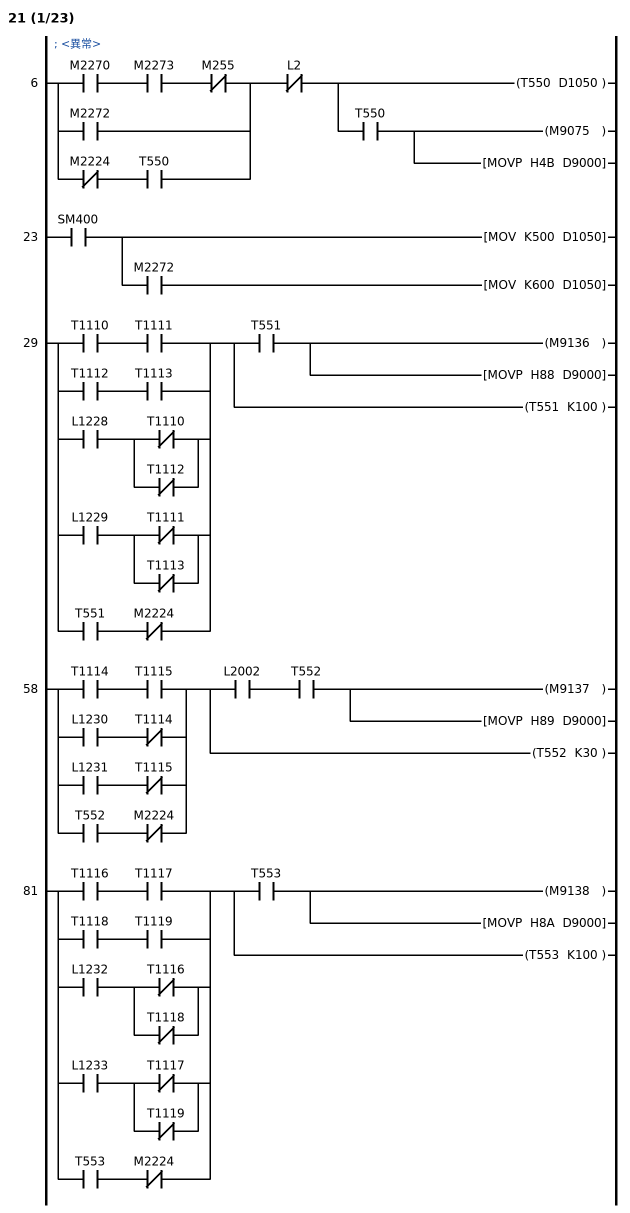
; <異常>
6     LD      M2270
      AND     M2273
      ANI     M255
      OR      M2272
      LDI     M2224
      AND     T550
      ORB
      ANI     L2
      OUT     T550 D1050
      AND     T550
      OUT     M9075
      MOVP    H4B D9000
23    LD      SM400
      MOV     K500 D1050
      AND     M2272
      MOV     K600 D1050
29    LD      T1110
      AND     T1111
      LD      T1112
      AND     T1113
      ORB
      LD      L1228
      LDI     T1110
      ORI     T1112
      ANB
      ORB
      LD      L1229
      LDI     T1111
      ORI     T1113
      ANB
      ORB
      LD      T551
      ANI     M2224
      ORB
      MPS
      AND     T551
      OUT     M9136
      MOVP    H88 D9000
      MPP
      OUT     T551 K100
58    LD      T1114
      AND     T1115
      LD      L1230
      ANI     T1114
      ORB
      LD      L1231
      ANI     T1115
      ORB
      LD      T552
      ANI     M2224
      ORB
      MPS
      AND     L2002
      AND     T552
      OUT     M9137
      MOVP    H89 D9000
      MPP
      OUT     T552 K30
81    LD      T1116
      AND     T1117
      LD      T1118
      AND     T1119
      ORB
      LD      L1232
      LDI     T1116
      ORI     T1118
      ANB
      ORB
      LD      L1233
      LDI     T1117
      ORI     T1119
      ANB
      ORB
      LD      T553
      ANI     M2224
      ORB
      MPS
      AND     T553
      OUT     M9138
      MOVP    H8A D9000
      MPP
      OUT     T553 K100
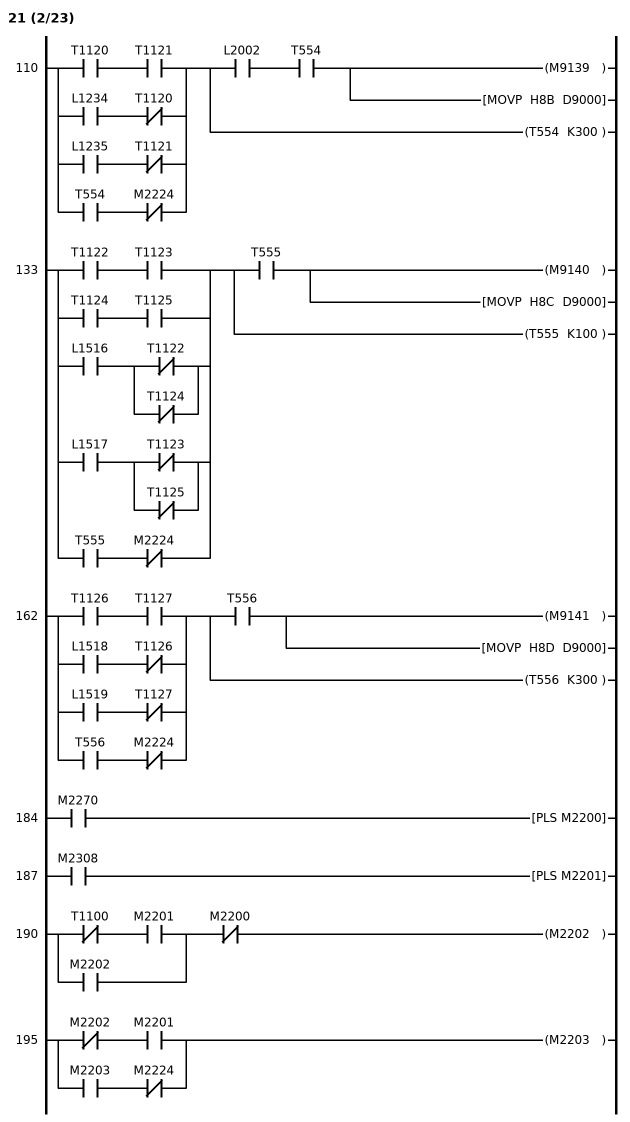
110   LD      T1120
      AND     T1121
      LD      L1234
      ANI     T1120
      ORB
      LD      L1235
      ANI     T1121
      ORB
      LD      T554
      ANI     M2224
      ORB
      MPS
      AND     L2002
      AND     T554
      OUT     M9139
      MOVP    H8B D9000
      MPP
      OUT     T554 K300
133   LD      T1122
      AND     T1123
      LD      T1124
      AND     T1125
      ORB
      LD      L1516
      LDI     T1122
      ORI     T1124
      ANB
      ORB
      LD      L1517
      LDI     T1123
      ORI     T1125
      ANB
      ORB
      LD      T555
      ANI     M2224
      ORB
      MPS
      AND     T555
      OUT     M9140
      MOVP    H8C D9000
      MPP
      OUT     T555 K100
162   LD      T1126
      AND     T1127
      LD      L1518
      ANI     T1126
      ORB
      LD      L1519
      ANI     T1127
      ORB
      LD      T556
      ANI     M2224
      ORB
      MPS
      AND     T556
      OUT     M9141
      MOVP    H8D D9000
      MPP
      OUT     T556 K300
184   LD      M2270
      PLS     M2200
187   LD      M2308
      PLS     M2201
190   LDI     T1100
      AND     M2201
      OR      M2202
      ANI     M2200
      OUT     M2202
195   LDI     M2202
      AND     M2201
      LD      M2203
      ANI     M2224
      ORB
      OUT     M2203
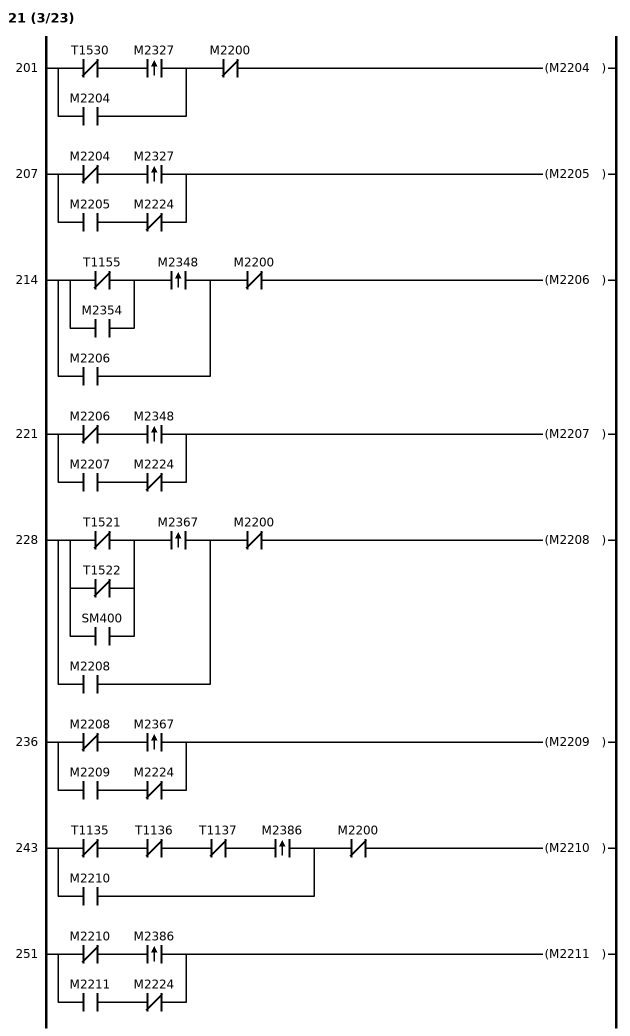
201   LDI     T1530
      ANDP    M2327
      OR      M2204
      ANI     M2200
      OUT     M2204
207   LDI     M2204
      ANDP    M2327
      LD      M2205
      ANI     M2224
      ORB
      OUT     M2205
214   LDI     T1155
      OR      M2354
      ANDP    M2348
      OR      M2206
      ANI     M2200
      OUT     M2206
221   LDI     M2206
      ANDP    M2348
      LD      M2207
      ANI     M2224
      ORB
      OUT     M2207
228   LDI     T1521
      ORI     T1522
      OR      SM400
      ANDP    M2367
      OR      M2208
      ANI     M2200
      OUT     M2208
236   LDI     M2208
      ANDP    M2367
      LD      M2209
      ANI     M2224
      ORB
      OUT     M2209
243   LDI     T1135
      ANI     T1136
      ANI     T1137
      ANDP    M2386
      OR      M2210
      ANI     M2200
      OUT     M2210
251   LDI     M2210
      ANDP    M2386
      LD      M2211
      ANI     M2224
      ORB
      OUT     M2211
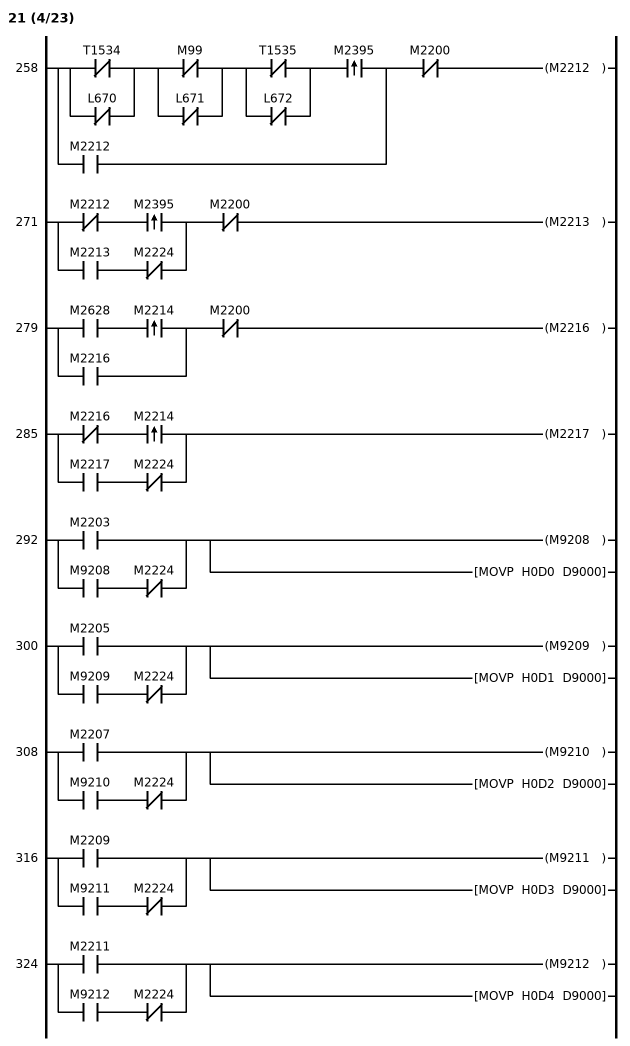
258   LDI     T1534
      ORI     L670
      LDI     M99
      ORI     L671
      ANB
      LDI     T1535
      ORI     L672
      ANB
      ANDP    M2395
      OR      M2212
      ANI     M2200
      OUT     M2212
271   LDI     M2212
      ANDP    M2395
      LD      M2213
      ANI     M2224
      ORB
      ANI     M2200
      OUT     M2213
279   LD      M2628
      ANDP    M2214
      OR      M2216
      ANI     M2200
      OUT     M2216
285   LDI     M2216
      ANDP    M2214
      LD      M2217
      ANI     M2224
      ORB
      OUT     M2217
292   LD      M2203
      LD      M9208
      ANI     M2224
      ORB
      OUT     M9208
      MOVP    H0D0 D9000
300   LD      M2205
      LD      M9209
      ANI     M2224
      ORB
      OUT     M9209
      MOVP    H0D1 D9000
308   LD      M2207
      LD      M9210
      ANI     M2224
      ORB
      OUT     M9210
      MOVP    H0D2 D9000
316   LD      M2209
      LD      M9211
      ANI     M2224
      ORB
      OUT     M9211
      MOVP    H0D3 D9000
324   LD      M2211
      LD      M9212
      ANI     M2224
      ORB
      OUT     M9212
      MOVP    H0D4 D9000
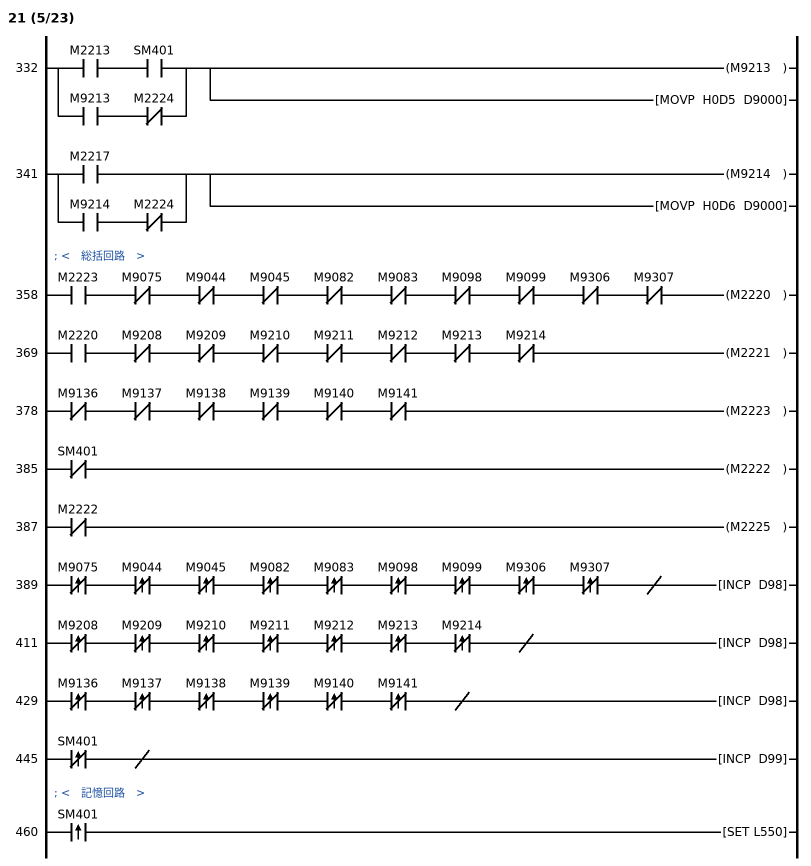
332   LD      M2213
      AND     SM401
      LD      M9213
      ANI     M2224
      ORB
      OUT     M9213
      MOVP    H0D5 D9000
341   LD      M2217
      LD      M9214
      ANI     M2224
      ORB
      OUT     M9214
      MOVP    H0D6 D9000
; <　総括回路　>
358   LD      M2223
      ANI     M9075
      ANI     M9044
      ANI     M9045
      ANI     M9082
      ANI     M9083
      ANI     M9098
      ANI     M9099
      ANI     M9306
      ANI     M9307
      OUT     M2220
369   LD      M2220
      ANI     M9208
      ANI     M9209
      ANI     M9210
      ANI     M9211
      ANI     M9212
      ANI     M9213
      ANI     M9214
      OUT     M2221
378   LDI     M9136
      ANI     M9137
      ANI     M9138
      ANI     M9139
      ANI     M9140
      ANI     M9141
      OUT     M2223
385   LDI     SM401
      OUT     M2222
387   LDI     M2222
      OUT     M2225
389   LDPI    M9075
      ANDPI   M9044
      ANDPI   M9045
      ANDPI   M9082
      ANDPI   M9083
      ANDPI   M9098
      ANDPI   M9099
      ANDPI   M9306
      ANDPI   M9307
      INV
      INCP    D98
411   LDPI    M9208
      ANDPI   M9209
      ANDPI   M9210
      ANDPI   M9211
      ANDPI   M9212
      ANDPI   M9213
      ANDPI   M9214
      INV
      INCP    D98
429   LDPI    M9136
      ANDPI   M9137
      ANDPI   M9138
      ANDPI   M9139
      ANDPI   M9140
      ANDPI   M9141
      INV
      INCP    D98
445   LDPI    SM401
      INV
      INCP    D99
; <　記憶回路　>
460   LDP     SM401
      SET     L550
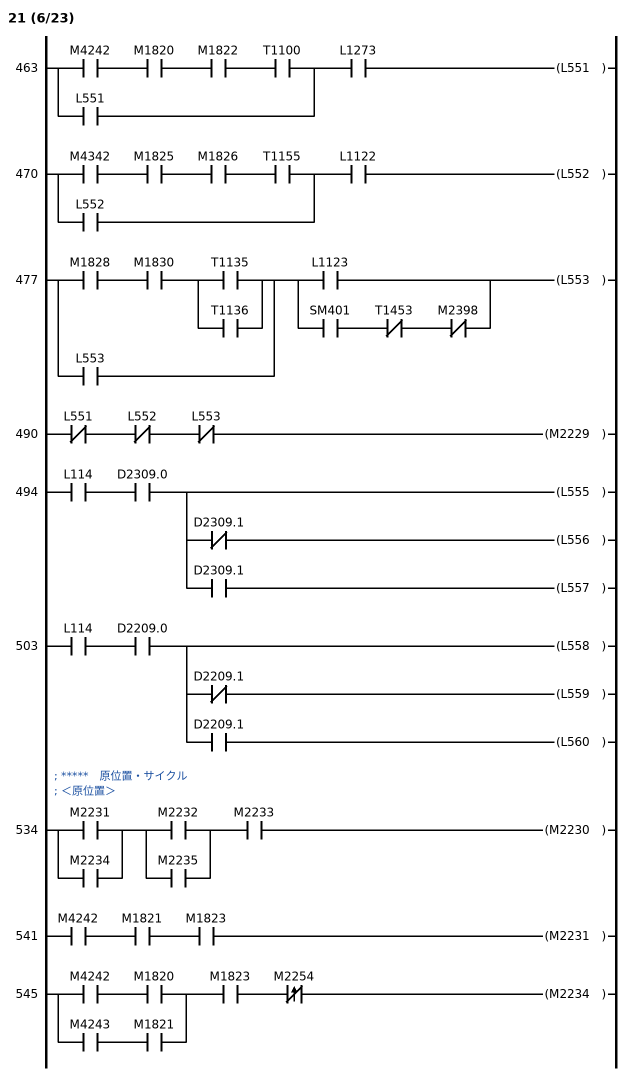
463   LD      M4242
      AND     M1820
      AND     M1822
      AND     T1100
      OR      L551
      AND     L1273
      OUT     L551
470   LD      M4342
      AND     M1825
      AND     M1826
      AND     T1155
      OR      L552
      AND     L1122
      OUT     L552
477   LD      M1828
      AND     M1830
      LD      T1135
      OR      T1136
      ANB
      OR      L553
      LD      L1123
      LD      SM401
      ANI     T1453
      ANI     M2398
      ORB
      ANB
      OUT     L553
490   LDI     L551
      ANI     L552
      ANI     L553
      OUT     M2229
494   LD      L114
      AND     D2309.0
      OUT     L555
      MPS
      ANI     D2309.1
      OUT     L556
      MPP
      AND     D2309.1
      OUT     L557
503   LD      L114
      AND     D2209.0
      OUT     L558
      MPS
      ANI     D2209.1
      OUT     L559
      MPP
      AND     D2209.1
      OUT     L560
; *****　原位置・サイクル
; ＜原位置＞
534   LD      M2231
      OR      M2234
      LD      M2232
      OR      M2235
      ANB
      AND     M2233
      OUT     M2230
541   LD      M4242
      AND     M1821
      AND     M1823
      OUT     M2231
545   LD      M4242
      AND     M1820
      LD      M4243
      AND     M1821
      ORB
      AND     M1823
      ANDPI   M2254
      OUT     M2234
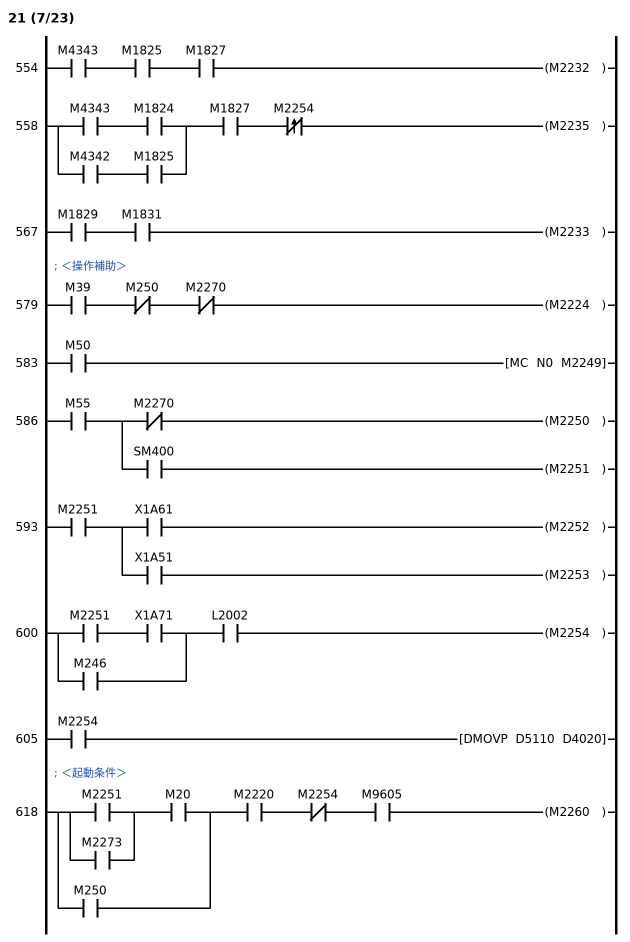
554   LD      M4343
      AND     M1825
      AND     M1827
      OUT     M2232
558   LD      M4343
      AND     M1824
      LD      M4342
      AND     M1825
      ORB
      AND     M1827
      ANDPI   M2254
      OUT     M2235
567   LD      M1829
      AND     M1831
      OUT     M2233
; ＜操作補助＞
579   LD      M39
      ANI     M250
      ANI     M2270
      OUT     M2224
583   LD      M50
      MC      N0 M2249
586   LD      M55
      MPS
      ANI     M2270
      OUT     M2250
      MPP
      AND     SM400
      OUT     M2251
593   LD      M2251
      MPS
      AND     X1A61
      OUT     M2252
      MPP
      AND     X1A51
      OUT     M2253
600   LD      M2251
      AND     X1A71
      OR      M246
      AND     L2002
      OUT     M2254
605   LD      M2254
      DMOVP   D5110 D4020
; ＜起動条件＞
618   LD      M2251
      OR      M2273
      AND     M20
      OR      M250
      AND     M2220
      ANI     M2254
      AND     M9605
      OUT     M2260
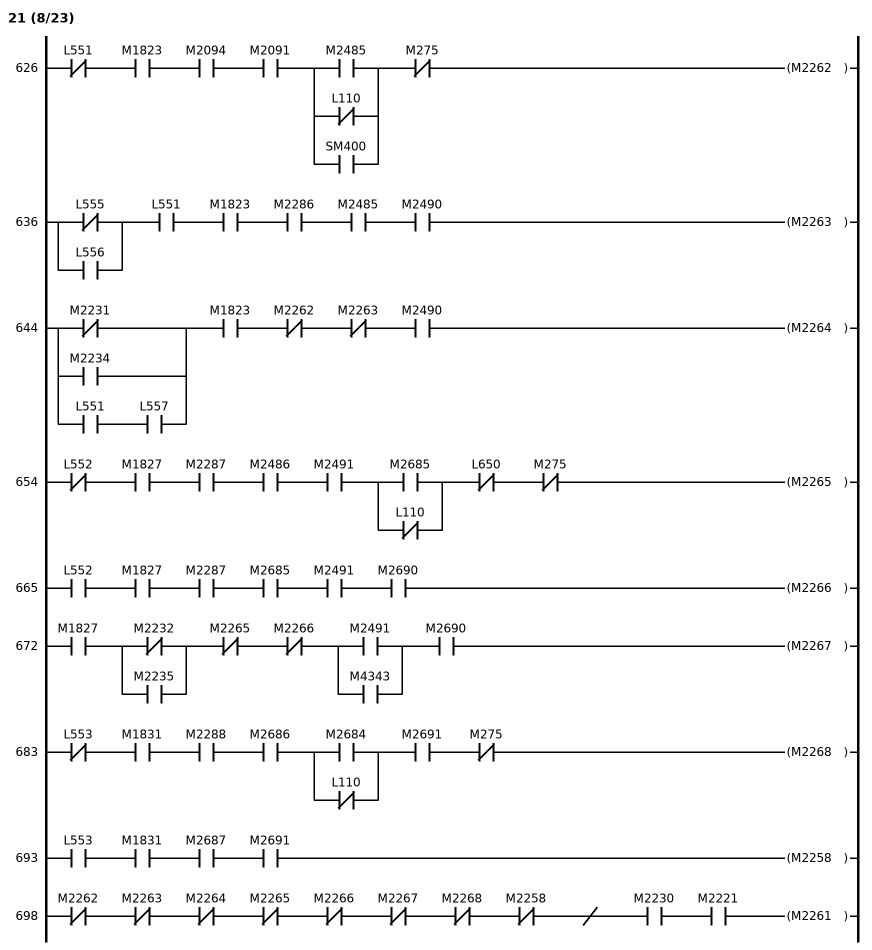
626   LDI     L551
      AND     M1823
      AND     M2094
      AND     M2091
      LD      M2485
      ORI     L110
      OR      SM400
      ANB
      ANI     M275
      OUT     M2262
636   LDI     L555
      OR      L556
      AND     L551
      AND     M1823
      AND     M2286
      AND     M2485
      AND     M2490
      OUT     M2263
644   LDI     M2231
      OR      M2234
      LD      L551
      AND     L557
      ORB
      AND     M1823
      ANI     M2262
      ANI     M2263
      AND     M2490
      OUT     M2264
654   LDI     L552
      AND     M1827
      AND     M2287
      AND     M2486
      AND     M2491
      LD      M2685
      ORI     L110
      ANB
      ANI     L650
      ANI     M275
      OUT     M2265
665   LD      L552
      AND     M1827
      AND     M2287
      AND     M2685
      AND     M2491
      AND     M2690
      OUT     M2266
672   LD      M1827
      LDI     M2232
      OR      M2235
      ANB
      ANI     M2265
      ANI     M2266
      LD      M2491
      OR      M4343
      ANB
      AND     M2690
      OUT     M2267
683   LDI     L553
      AND     M1831
      AND     M2288
      AND     M2686
      LD      M2684
      ORI     L110
      ANB
      AND     M2691
      ANI     M275
      OUT     M2268
693   LD      L553
      AND     M1831
      AND     M2687
      AND     M2691
      OUT     M2258
698   LDI     M2262
      ANI     M2263
      ANI     M2264
      ANI     M2265
      ANI     M2266
      ANI     M2267
      ANI     M2268
      ANI     M2258
      INV
      AND     M2230
      AND     M2221
      OUT     M2261
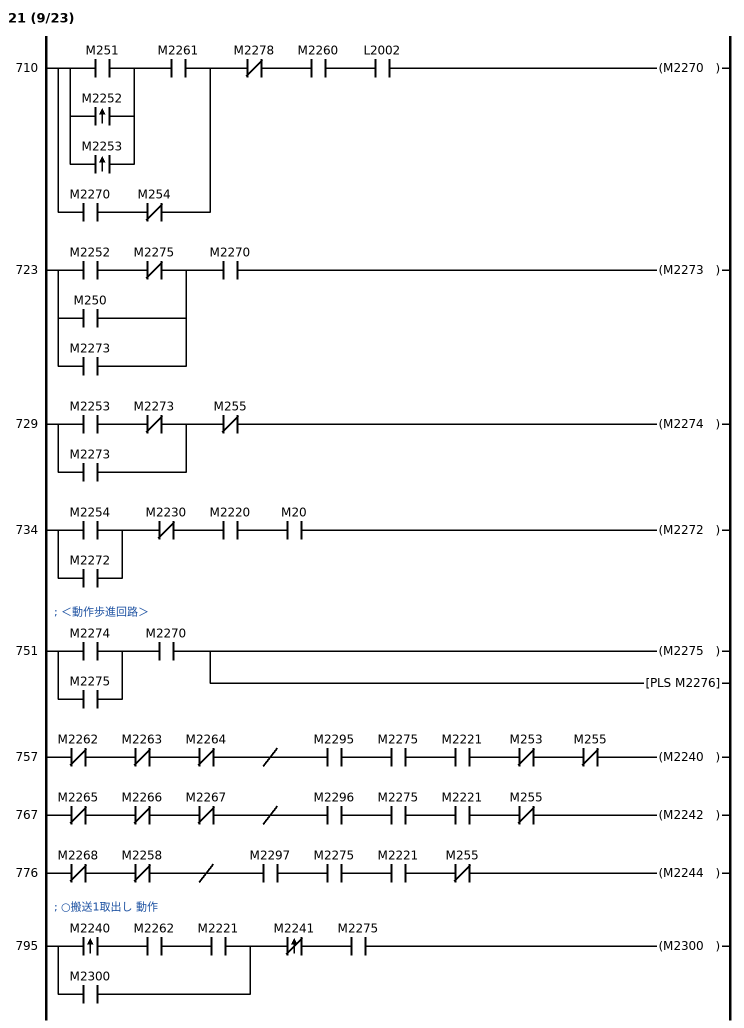
710   LD      M251
      ORP     M2252
      ORP     M2253
      AND     M2261
      LD      M2270
      ANI     M254
      ORB
      ANI     M2278
      AND     M2260
      AND     L2002
      OUT     M2270
723   LD      M2252
      ANI     M2275
      OR      M250
      OR      M2273
      AND     M2270
      OUT     M2273
729   LD      M2253
      ANI     M2273
      OR      M2273
      ANI     M255
      OUT     M2274
734   LD      M2254
      OR      M2272
      ANI     M2230
      AND     M2220
      AND     M20
      OUT     M2272
; ＜動作歩進回路＞
751   LD      M2274
      OR      M2275
      AND     M2270
      OUT     M2275
      PLS     M2276
757   LDI     M2262
      ANI     M2263
      ANI     M2264
      INV
      AND     M2295
      AND     M2275
      AND     M2221
      ANI     M253
      ANI     M255
      OUT     M2240
767   LDI     M2265
      ANI     M2266
      ANI     M2267
      INV
      AND     M2296
      AND     M2275
      AND     M2221
      ANI     M255
      OUT     M2242
776   LDI     M2268
      ANI     M2258
      INV
      AND     M2297
      AND     M2275
      AND     M2221
      ANI     M255
      OUT     M2244
; ○搬送1取出し 動作
795   LDP     M2240
      AND     M2262
      AND     M2221
      OR      M2300
      ANDPI   M2241
      AND     M2275
      OUT     M2300
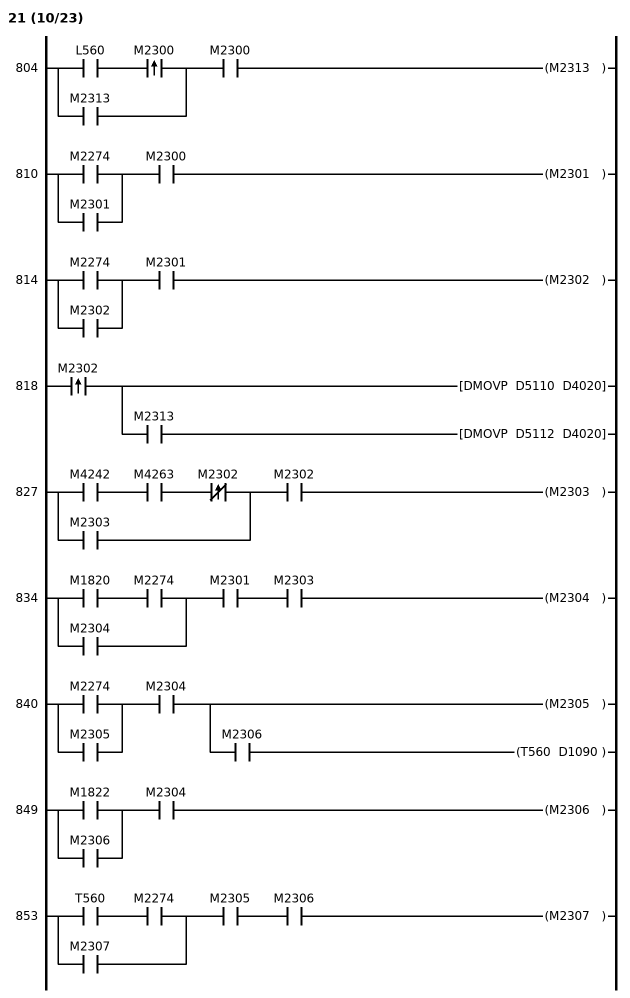
804   LD      L560
      ANDP    M2300
      OR      M2313
      AND     M2300
      OUT     M2313
810   LD      M2274
      OR      M2301
      AND     M2300
      OUT     M2301
814   LD      M2274
      OR      M2302
      AND     M2301
      OUT     M2302
818   LDP     M2302
      DMOVP   D5110 D4020
      AND     M2313
      DMOVP   D5112 D4020
827   LD      M4242
      AND     M4263
      ANDPI   M2302
      OR      M2303
      AND     M2302
      OUT     M2303
834   LD      M1820
      AND     M2274
      OR      M2304
      AND     M2301
      AND     M2303
      OUT     M2304
840   LD      M2274
      OR      M2305
      AND     M2304
      OUT     M2305
      AND     M2306
      OUT     T560 D1090
849   LD      M1822
      OR      M2306
      AND     M2304
      OUT     M2306
853   LD      T560
      AND     M2274
      OR      M2307
      AND     M2305
      AND     M2306
      OUT     M2307
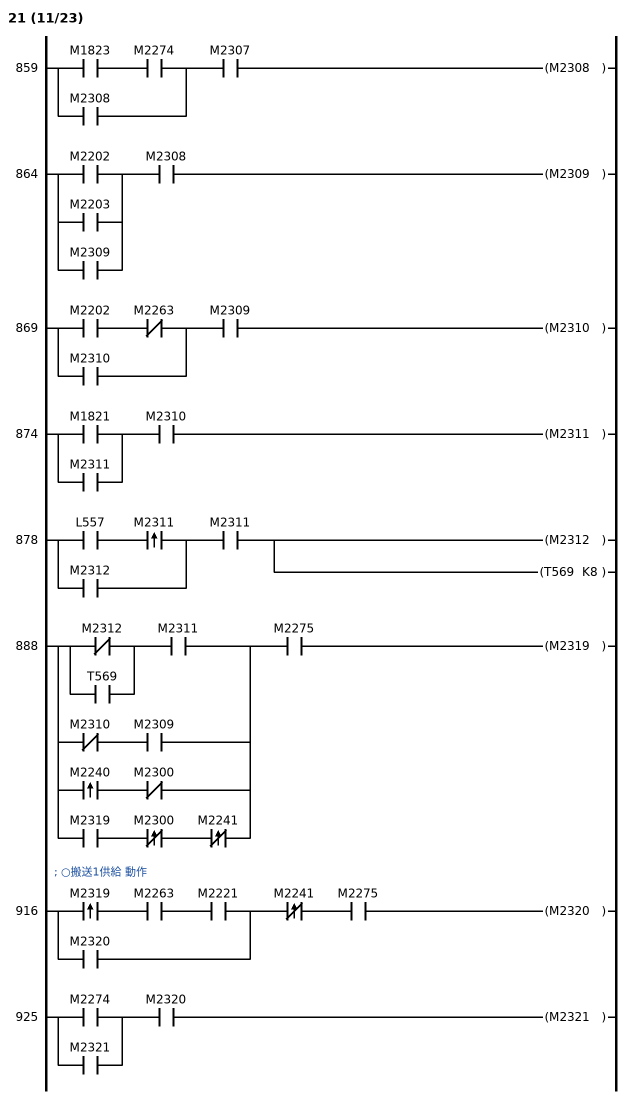
859   LD      M1823
      AND     M2274
      OR      M2308
      AND     M2307
      OUT     M2308
864   LD      M2202
      OR      M2203
      OR      M2309
      AND     M2308
      OUT     M2309
869   LD      M2202
      ANI     M2263
      OR      M2310
      AND     M2309
      OUT     M2310
874   LD      M1821
      OR      M2311
      AND     M2310
      OUT     M2311
878   LD      L557
      ANDP    M2311
      OR      M2312
      AND     M2311
      OUT     M2312
      OUT     T569 K8
888   LDI     M2312
      OR      T569
      AND     M2311
      LDI     M2310
      AND     M2309
      ORB
      LDP     M2240
      ANI     M2300
      ORB
      LD      M2319
      ANDPI   M2300
      ANDPI   M2241
      ORB
      AND     M2275
      OUT     M2319
; ○搬送1供給 動作
916   LDP     M2319
      AND     M2263
      AND     M2221
      OR      M2320
      ANDPI   M2241
      AND     M2275
      OUT     M2320
925   LD      M2274
      OR      M2321
      AND     M2320
      OUT     M2321
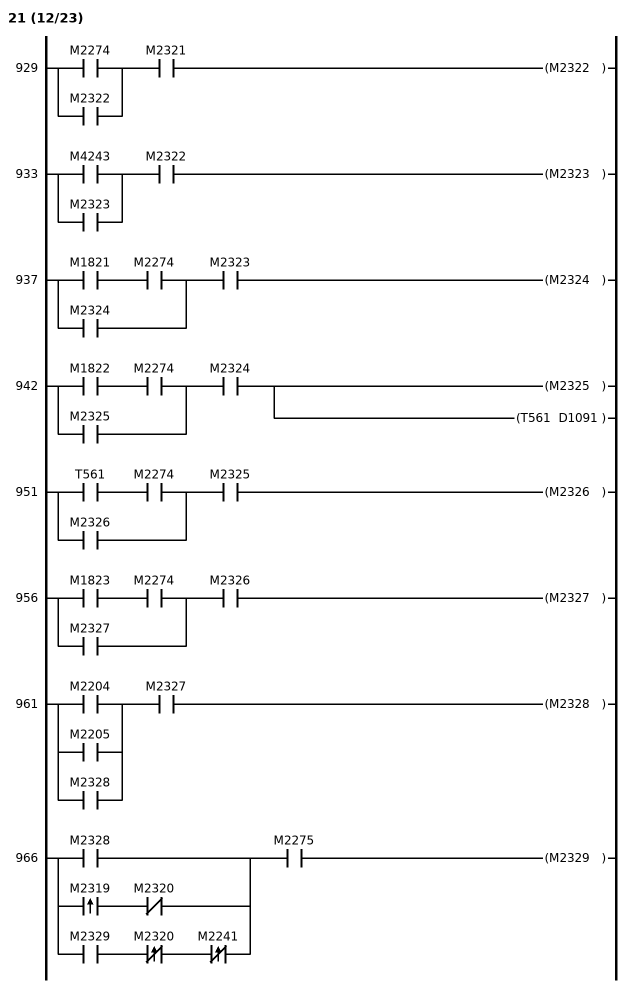
929   LD      M2274
      OR      M2322
      AND     M2321
      OUT     M2322
933   LD      M4243
      OR      M2323
      AND     M2322
      OUT     M2323
937   LD      M1821
      AND     M2274
      OR      M2324
      AND     M2323
      OUT     M2324
942   LD      M1822
      AND     M2274
      OR      M2325
      AND     M2324
      OUT     M2325
      OUT     T561 D1091
951   LD      T561
      AND     M2274
      OR      M2326
      AND     M2325
      OUT     M2326
956   LD      M1823
      AND     M2274
      OR      M2327
      AND     M2326
      OUT     M2327
961   LD      M2204
      OR      M2205
      OR      M2328
      AND     M2327
      OUT     M2328
966   LD      M2328
      LDP     M2319
      ANI     M2320
      ORB
      LD      M2329
      ANDPI   M2320
      ANDPI   M2241
      ORB
      AND     M2275
      OUT     M2329
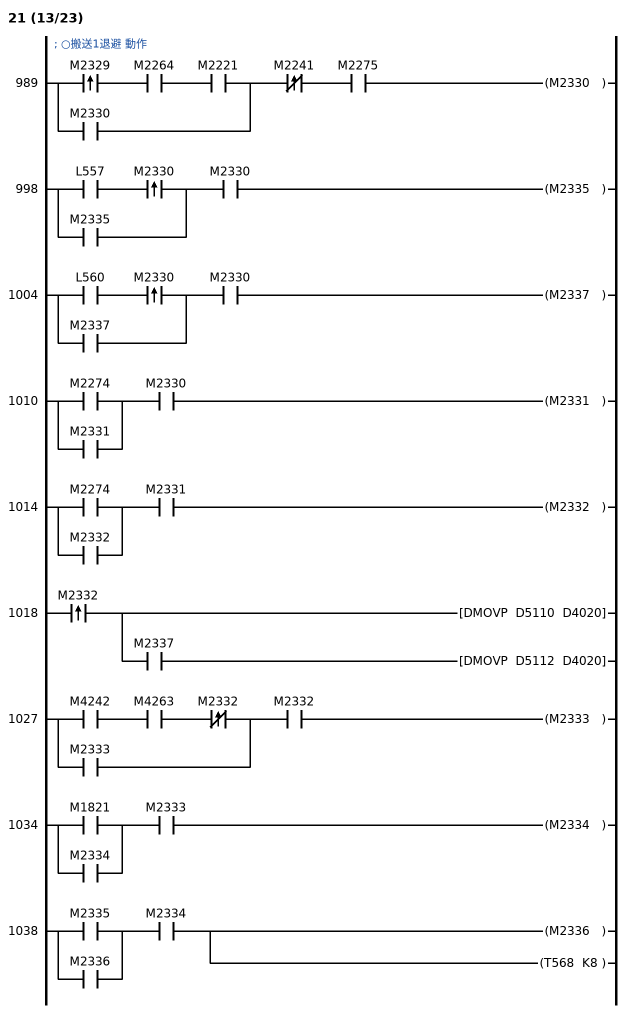
; ○搬送1退避 動作
989   LDP     M2329
      AND     M2264
      AND     M2221
      OR      M2330
      ANDPI   M2241
      AND     M2275
      OUT     M2330
998   LD      L557
      ANDP    M2330
      OR      M2335
      AND     M2330
      OUT     M2335
1004  LD      L560
      ANDP    M2330
      OR      M2337
      AND     M2330
      OUT     M2337
1010  LD      M2274
      OR      M2331
      AND     M2330
      OUT     M2331
1014  LD      M2274
      OR      M2332
      AND     M2331
      OUT     M2332
1018  LDP     M2332
      DMOVP   D5110 D4020
      AND     M2337
      DMOVP   D5112 D4020
1027  LD      M4242
      AND     M4263
      ANDPI   M2332
      OR      M2333
      AND     M2332
      OUT     M2333
1034  LD      M1821
      OR      M2334
      AND     M2333
      OUT     M2334
1038  LD      M2335
      OR      M2336
      AND     M2334
      OUT     M2336
      OUT     T568 K8
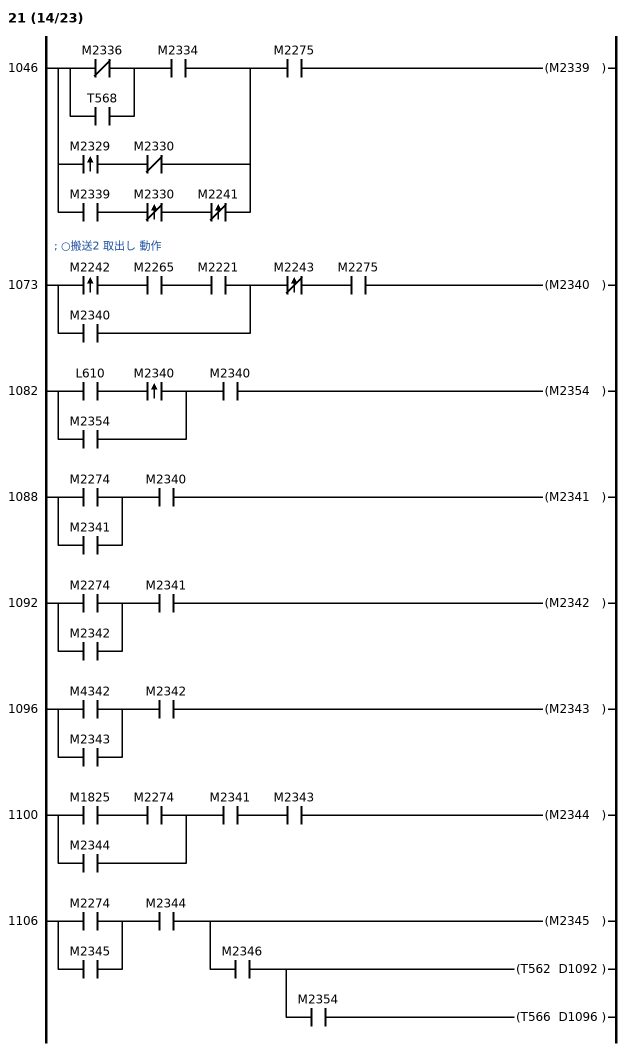
1046  LDI     M2336
      OR      T568
      AND     M2334
      LDP     M2329
      ANI     M2330
      ORB
      LD      M2339
      ANDPI   M2330
      ANDPI   M2241
      ORB
      AND     M2275
      OUT     M2339
; ○搬送2 取出し 動作
1073  LDP     M2242
      AND     M2265
      AND     M2221
      OR      M2340
      ANDPI   M2243
      AND     M2275
      OUT     M2340
1082  LD      L610
      ANDP    M2340
      OR      M2354
      AND     M2340
      OUT     M2354
1088  LD      M2274
      OR      M2341
      AND     M2340
      OUT     M2341
1092  LD      M2274
      OR      M2342
      AND     M2341
      OUT     M2342
1096  LD      M4342
      OR      M2343
      AND     M2342
      OUT     M2343
1100  LD      M1825
      AND     M2274
      OR      M2344
      AND     M2341
      AND     M2343
      OUT     M2344
1106  LD      M2274
      OR      M2345
      AND     M2344
      OUT     M2345
      AND     M2346
      OUT     T562 D1092
      AND     M2354
      OUT     T566 D1096
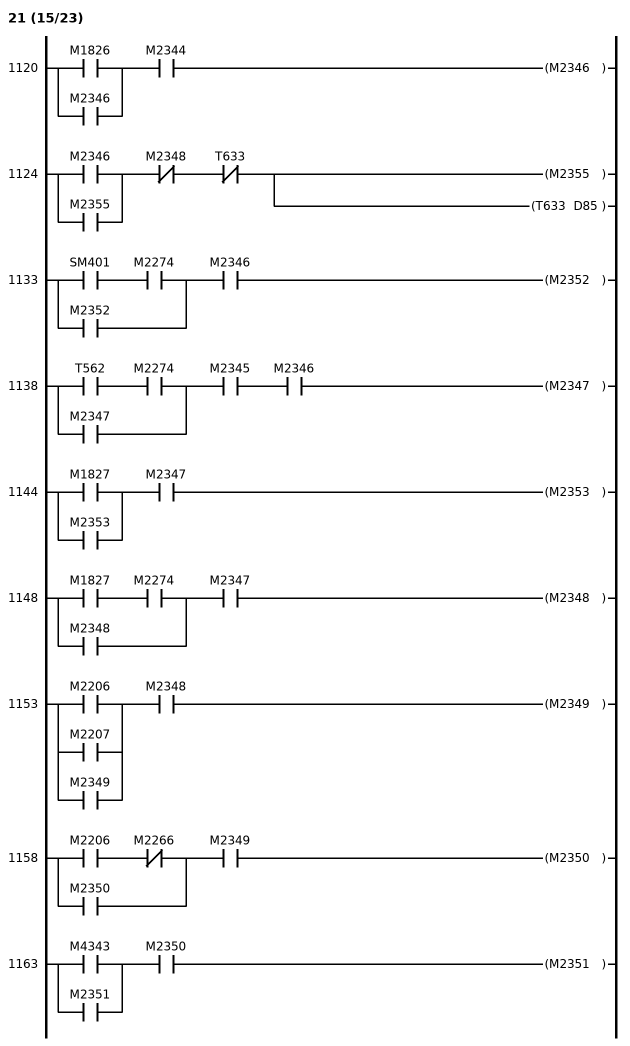
1120  LD      M1826
      OR      M2346
      AND     M2344
      OUT     M2346
1124  LD      M2346
      OR      M2355
      ANI     M2348
      ANI     T633
      OUT     M2355
      OUT     T633 D85
1133  LD      SM401
      AND     M2274
      OR      M2352
      AND     M2346
      OUT     M2352
1138  LD      T562
      AND     M2274
      OR      M2347
      AND     M2345
      AND     M2346
      OUT     M2347
1144  LD      M1827
      OR      M2353
      AND     M2347
      OUT     M2353
1148  LD      M1827
      AND     M2274
      OR      M2348
      AND     M2347
      OUT     M2348
1153  LD      M2206
      OR      M2207
      OR      M2349
      AND     M2348
      OUT     M2349
1158  LD      M2206
      ANI     M2266
      OR      M2350
      AND     M2349
      OUT     M2350
1163  LD      M4343
      OR      M2351
      AND     M2350
      OUT     M2351
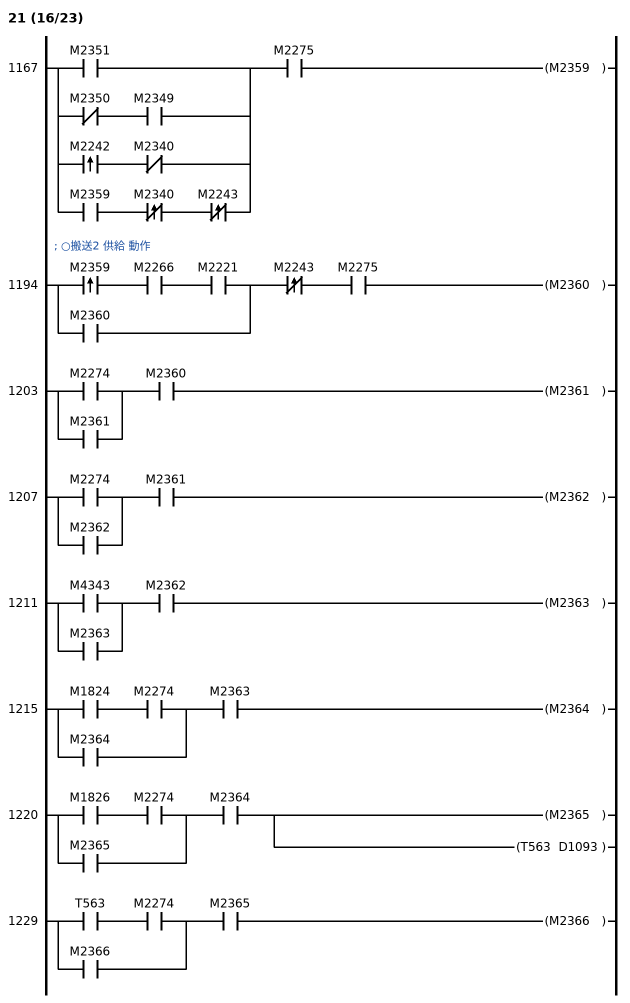
1167  LD      M2351
      LDI     M2350
      AND     M2349
      ORB
      LDP     M2242
      ANI     M2340
      ORB
      LD      M2359
      ANDPI   M2340
      ANDPI   M2243
      ORB
      AND     M2275
      OUT     M2359
; ○搬送2 供給 動作
1194  LDP     M2359
      AND     M2266
      AND     M2221
      OR      M2360
      ANDPI   M2243
      AND     M2275
      OUT     M2360
1203  LD      M2274
      OR      M2361
      AND     M2360
      OUT     M2361
1207  LD      M2274
      OR      M2362
      AND     M2361
      OUT     M2362
1211  LD      M4343
      OR      M2363
      AND     M2362
      OUT     M2363
1215  LD      M1824
      AND     M2274
      OR      M2364
      AND     M2363
      OUT     M2364
1220  LD      M1826
      AND     M2274
      OR      M2365
      AND     M2364
      OUT     M2365
      OUT     T563 D1093
1229  LD      T563
      AND     M2274
      OR      M2366
      AND     M2365
      OUT     M2366
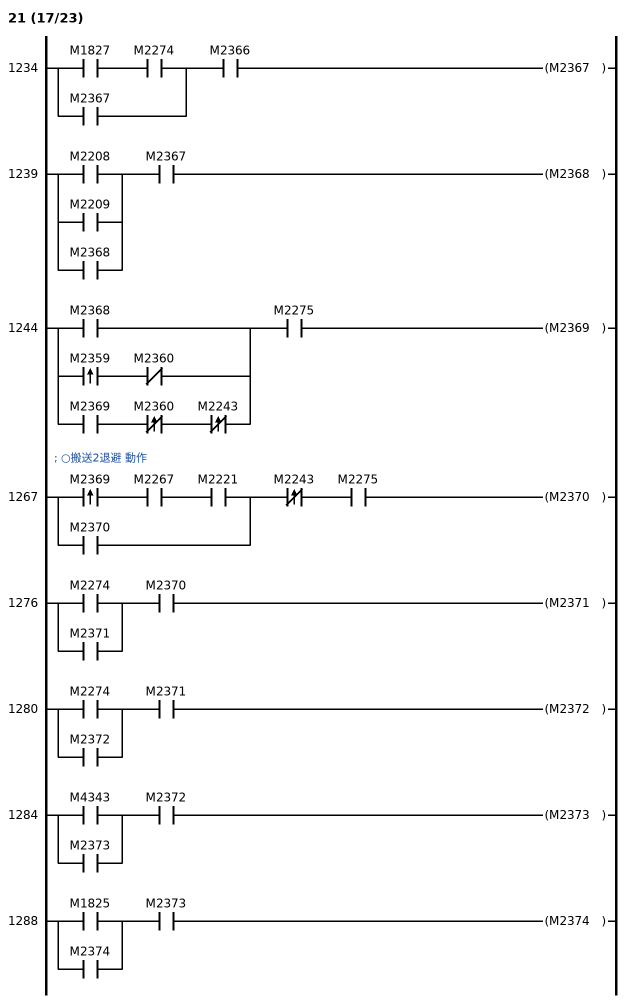
1234  LD      M1827
      AND     M2274
      OR      M2367
      AND     M2366
      OUT     M2367
1239  LD      M2208
      OR      M2209
      OR      M2368
      AND     M2367
      OUT     M2368
1244  LD      M2368
      LDP     M2359
      ANI     M2360
      ORB
      LD      M2369
      ANDPI   M2360
      ANDPI   M2243
      ORB
      AND     M2275
      OUT     M2369
; ○搬送2退避 動作
1267  LDP     M2369
      AND     M2267
      AND     M2221
      OR      M2370
      ANDPI   M2243
      AND     M2275
      OUT     M2370
1276  LD      M2274
      OR      M2371
      AND     M2370
      OUT     M2371
1280  LD      M2274
      OR      M2372
      AND     M2371
      OUT     M2372
1284  LD      M4343
      OR      M2373
      AND     M2372
      OUT     M2373
1288  LD      M1825
      OR      M2374
      AND     M2373
      OUT     M2374
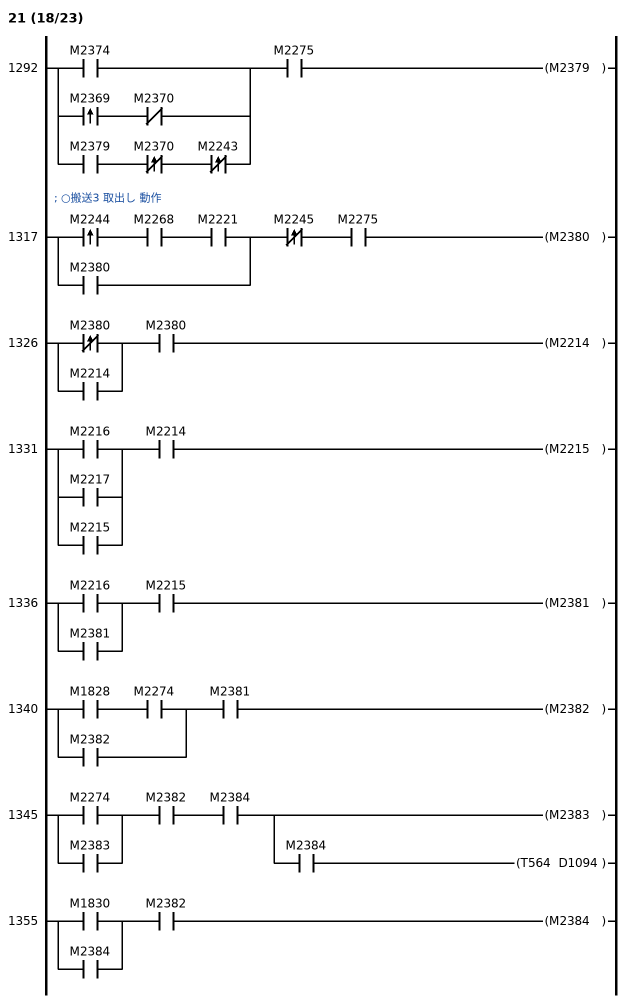
1292  LD      M2374
      LDP     M2369
      ANI     M2370
      ORB
      LD      M2379
      ANDPI   M2370
      ANDPI   M2243
      ORB
      AND     M2275
      OUT     M2379
; ○搬送3 取出し 動作
1317  LDP     M2244
      AND     M2268
      AND     M2221
      OR      M2380
      ANDPI   M2245
      AND     M2275
      OUT     M2380
1326  LDPI    M2380
      OR      M2214
      AND     M2380
      OUT     M2214
1331  LD      M2216
      OR      M2217
      OR      M2215
      AND     M2214
      OUT     M2215
1336  LD      M2216
      OR      M2381
      AND     M2215
      OUT     M2381
1340  LD      M1828
      AND     M2274
      OR      M2382
      AND     M2381
      OUT     M2382
1345  LD      M2274
      OR      M2383
      AND     M2382
      AND     M2384
      OUT     M2383
      AND     M2384
      OUT     T564 D1094
1355  LD      M1830
      OR      M2384
      AND     M2382
      OUT     M2384
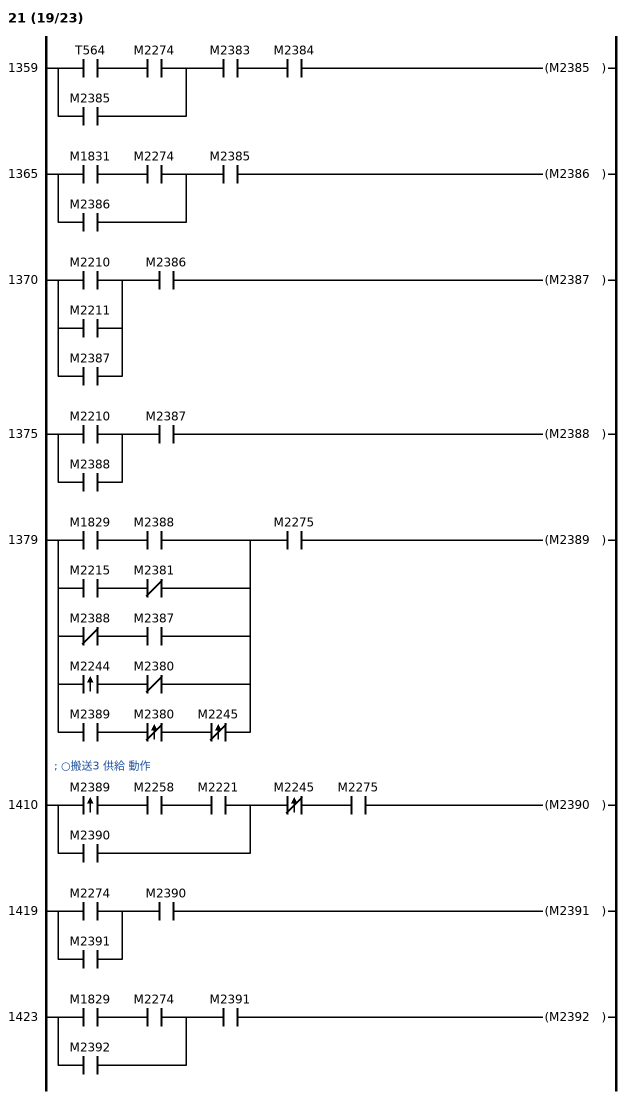
1359  LD      T564
      AND     M2274
      OR      M2385
      AND     M2383
      AND     M2384
      OUT     M2385
1365  LD      M1831
      AND     M2274
      OR      M2386
      AND     M2385
      OUT     M2386
1370  LD      M2210
      OR      M2211
      OR      M2387
      AND     M2386
      OUT     M2387
1375  LD      M2210
      OR      M2388
      AND     M2387
      OUT     M2388
1379  LD      M1829
      AND     M2388
      LD      M2215
      ANI     M2381
      ORB
      LDI     M2388
      AND     M2387
      ORB
      LDP     M2244
      ANI     M2380
      ORB
      LD      M2389
      ANDPI   M2380
      ANDPI   M2245
      ORB
      AND     M2275
      OUT     M2389
; ○搬送3 供給 動作
1410  LDP     M2389
      AND     M2258
      AND     M2221
      OR      M2390
      ANDPI   M2245
      AND     M2275
      OUT     M2390
1419  LD      M2274
      OR      M2391
      AND     M2390
      OUT     M2391
1423  LD      M1829
      AND     M2274
      OR      M2392
      AND     M2391
      OUT     M2392
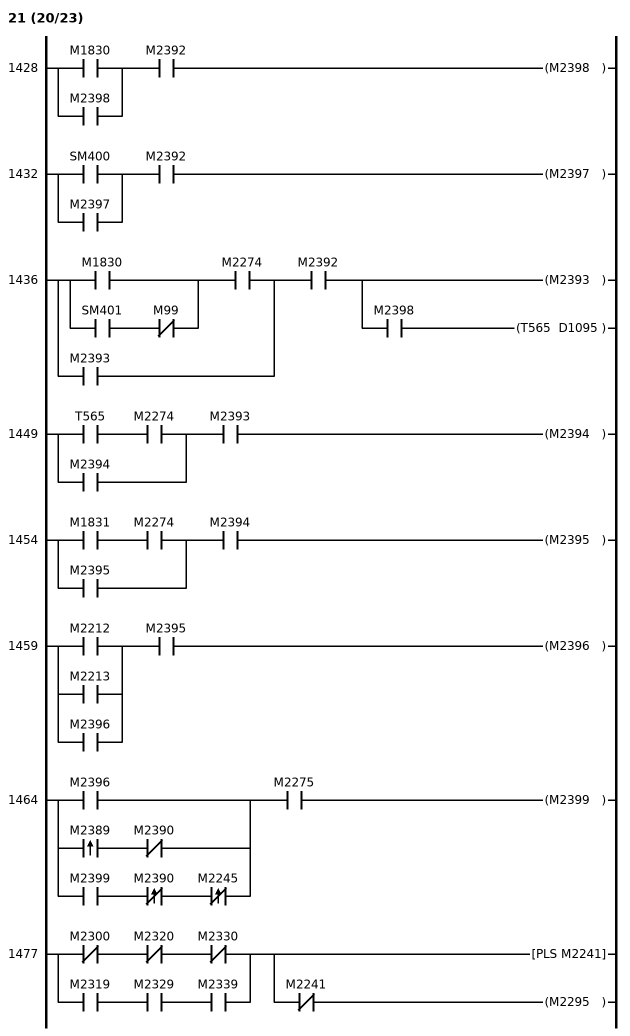
1428  LD      M1830
      OR      M2398
      AND     M2392
      OUT     M2398
1432  LD      SM400
      OR      M2397
      AND     M2392
      OUT     M2397
1436  LD      M1830
      LD      SM401
      ANI     M99
      ORB
      AND     M2274
      OR      M2393
      AND     M2392
      OUT     M2393
      AND     M2398
      OUT     T565 D1095
1449  LD      T565
      AND     M2274
      OR      M2394
      AND     M2393
      OUT     M2394
1454  LD      M1831
      AND     M2274
      OR      M2395
      AND     M2394
      OUT     M2395
1459  LD      M2212
      OR      M2213
      OR      M2396
      AND     M2395
      OUT     M2396
1464  LD      M2396
      LDP     M2389
      ANI     M2390
      ORB
      LD      M2399
      ANDPI   M2390
      ANDPI   M2245
      ORB
      AND     M2275
      OUT     M2399
1477  LDI     M2300
      ANI     M2320
      ANI     M2330
      LD      M2319
      AND     M2329
      AND     M2339
      ORB
      PLS     M2241
      ANI     M2241
      OUT     M2295
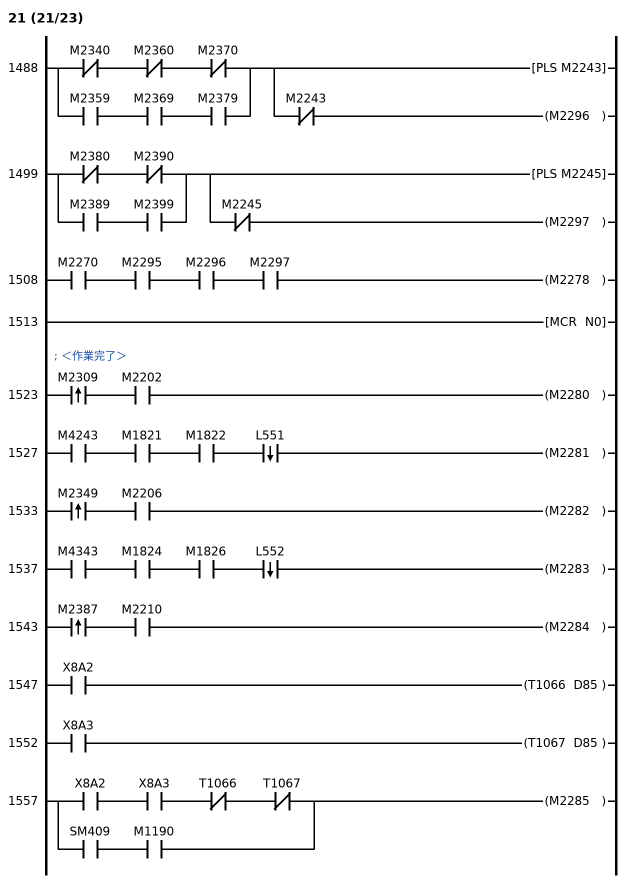
1488  LDI     M2340
      ANI     M2360
      ANI     M2370
      LD      M2359
      AND     M2369
      AND     M2379
      ORB
      PLS     M2243
      ANI     M2243
      OUT     M2296
1499  LDI     M2380
      ANI     M2390
      LD      M2389
      AND     M2399
      ORB
      PLS     M2245
      ANI     M2245
      OUT     M2297
1508  LD      M2270
      AND     M2295
      AND     M2296
      AND     M2297
      OUT     M2278
1513  MCR     N0
; ＜作業完了＞
1523  LDP     M2309
      AND     M2202
      OUT     M2280
1527  LD      M4243
      AND     M1821
      AND     M1822
      ANDF    L551
      OUT     M2281
1533  LDP     M2349
      AND     M2206
      OUT     M2282
1537  LD      M4343
      AND     M1824
      AND     M1826
      ANDF    L552
      OUT     M2283
1543  LDP     M2387
      AND     M2210
      OUT     M2284
1547  LD      X8A2
      OUT     T1066 D85
1552  LD      X8A3
      OUT     T1067 D85
1557  LD      X8A2
      AND     X8A3
      ANI     T1066
      ANI     T1067
      LD      SM409
      AND     M1190
      ORB
      OUT     M2285
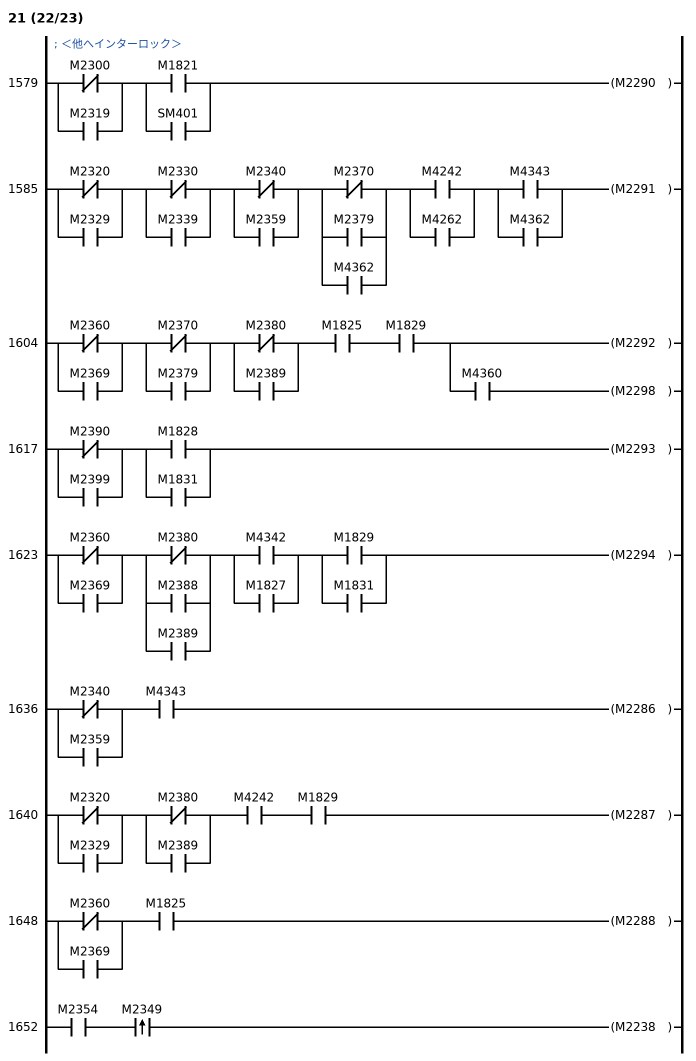
; ＜他へインターロック＞
1579  LDI     M2300
      OR      M2319
      LD      M1821
      OR      SM401
      ANB
      OUT     M2290
1585  LDI     M2320
      OR      M2329
      LDI     M2330
      OR      M2339
      ANB
      LDI     M2340
      OR      M2359
      ANB
      LDI     M2370
      OR      M2379
      OR      M4362
      ANB
      LD      M4242
      OR      M4262
      ANB
      LD      M4343
      OR      M4362
      ANB
      OUT     M2291
1604  LDI     M2360
      OR      M2369
      LDI     M2370
      OR      M2379
      ANB
      LDI     M2380
      OR      M2389
      ANB
      AND     M1825
      AND     M1829
      OUT     M2292
      AND     M4360
      OUT     M2298
1617  LDI     M2390
      OR      M2399
      LD      M1828
      OR      M1831
      ANB
      OUT     M2293
1623  LDI     M2360
      OR      M2369
      LDI     M2380
      OR      M2388
      OR      M2389
      ANB
      LD      M4342
      OR      M1827
      ANB
      LD      M1829
      OR      M1831
      ANB
      OUT     M2294
1636  LDI     M2340
      OR      M2359
      AND     M4343
      OUT     M2286
1640  LDI     M2320
      OR      M2329
      LDI     M2380
      OR      M2389
      ANB
      AND     M4242
      AND     M1829
      OUT     M2287
1648  LDI     M2360
      OR      M2369
      AND     M1825
      OUT     M2288
1652  LD      M2354
      ANDP    M2349
      OUT     M2238
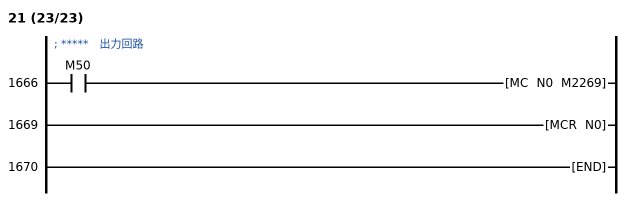
; *****　出力回路
1666  LD      M50
      MC      N0 M2269
1669  MCR     N0
1670  END
END_PROGRAM

PROGRAM 22
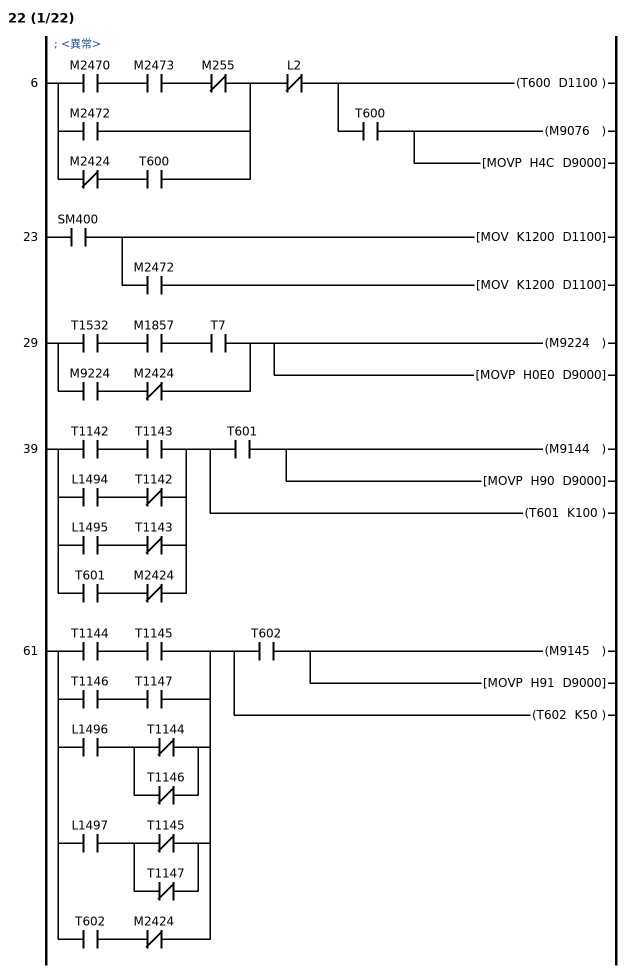
; <異常>
6     LD      M2470
      AND     M2473
      ANI     M255
      OR      M2472
      LDI     M2424
      AND     T600
      ORB
      ANI     L2
      OUT     T600 D1100
      AND     T600
      OUT     M9076
      MOVP    H4C D9000
23    LD      SM400
      MOV     K1200 D1100
      AND     M2472
      MOV     K1200 D1100
29    LD      T1532
      AND     M1857
      AND     T7
      LD      M9224
      ANI     M2424
      ORB
      OUT     M9224
      MOVP    H0E0 D9000
39    LD      T1142
      AND     T1143
      LD      L1494
      ANI     T1142
      ORB
      LD      L1495
      ANI     T1143
      ORB
      LD      T601
      ANI     M2424
      ORB
      MPS
      AND     T601
      OUT     M9144
      MOVP    H90 D9000
      MPP
      OUT     T601 K100
61    LD      T1144
      AND     T1145
      LD      T1146
      AND     T1147
      ORB
      LD      L1496
      LDI     T1144
      ORI     T1146
      ANB
      ORB
      LD      L1497
      LDI     T1145
      ORI     T1147
      ANB
      ORB
      LD      T602
      ANI     M2424
      ORB
      MPS
      AND     T602
      OUT     M9145
      MOVP    H91 D9000
      MPP
      OUT     T602 K50
